// TIA Portal V16 export
// export: Created 2023-03-29T11:03:19.8804357Z, ExportSetting WithDefaults, DisplayName Totally Integrated Automation Portal, DisplayVersion V16 Update 6, DisplayName TIA Portal Version Control Interface, DisplayVersion V16 Update 2, DisplayName TIA Portal Openness, DisplayVersion V16 Update 6, DisplayName STEP 7 Professional, DisplayVersion V16 Update 6, DisplayName STEP 7 Safety, DisplayVersion V16, DisplayName WinCC Advanced, DisplayVersion V16 Update 6
DATA_BLOCK "DB10_instance_SCADA"   // DB10
TITLE = SCADA
{ S7_Optimized_Access := 'FALSE' }
AUTHOR : rtecmer
VERSION : 0.1
// stored: AutoNumber false, DBAccessibleFromOPCUA true, IsOnlyStoredInLoadMemory false, IsWriteProtectedInAS false
   VAR
      Clock : Time;
      Watchdog : Int;
      instZ1 : Word := 33924;   // status zasuwy
      instZ2 : Word := 33924;   // status zasuwy
      instZ3 : Word := 33924;   // status zasuwy
      instZ4 : Word := 33924;   // status zasuwy
      instZ5 : Word := 33924;   // status zasuwy
      instZ6 : Word := 33924;   // status zasuwy
      instZ7 : Word := 33924;   // status zasuwy
      instZ8 : Word := 33924;   // status zasuwy
      instZ9 : Word := 33924;   // status zasuwy
      instZ10 : Word := 33924;   // status zasuwy
      actPoziomZbiornik_1 : Real;   // aktualny poziom w zbirniku
      actPoziomZbiornik_2 : Real := 0.0;   // aktualny poziom w zbirniku
      actPoziomZbiornik_3 : Real := 0.0;   // aktualny poziom w zbirniku
      actPoziomZbiornik_4 : Real := 0.0;   // aktualny poziom w zbirniku
      actPoziomZbiornik_5 : Real := 0.0;   // aktualny poziom w zbirniku
      actPrzepływ_Q2 : Real;   // aktualny przepływ Q2 - studnia pomiarowa przed pompownią
      sumPrzepływVF_Q2 : Real;   // suma przepływu
      statusPrzepływVR_Q2 : Real := 0.0;   // status przepływomierza
      setPołożenieZ10 : Word := 40;   // zadany [%] otwarcia
      actPołożenieZ10 : Word;   // aktualny [%] otwarcia
      rtu_mpp04_2error_status : Word;   // status błędu modbus przepływomierz Q2
      ModelSterowania : Word;   // Sygnały sterowania strategią pompownia - 0= wyłaczone, 1=dosilanie, 2=przetłaczanie,3=automat, 4=ręczne
      TrybSterowania : Word;   // Tryb 0-wyłączony, 1- Dobowy, 2- Tygodniowy, 3-Ręczny
      "Alarms only" : Word;   // Instancja alarmów (bit 68.0 - Error komunikacji z HMI)
      setPoziomNapełniania : Real := 550.0;   // zadana wartość napełniania
      setPoziomOpróżnianai : Real := 30.0;   // zadana wartość opróżniania
      "actCiśnienie-magistralaB5" : Real := 6.6;   // ciśnienie na przewodzie zasilania 9magistrala)
      rtu_step_reset : Bool;   // reset modbus RTU
      actTime_FillingOn : Real;   // godzina start napełnianie
      actTime_FillingOff : Real;   // godzina stop napełnianie
      actTime_EptyingOn : Real;   // godzina start przetłaczanie
      actTime_EptyingOff : Real;   // godzina stop przetłaczanie
      actTime : Real;   // czas aktualny
      actDTL_FillingOn : DTL := DTL#2022-08-02-00:05:00;   // zmienna DTL napełnianie start
      actDTL_FillingOff : DTL := DTL#2022-08-02-17:00:00.000000003;   // zmienna DTL napełnianie stop
      actDTL_pumpingOn : DTL := DTL#2022-08-02-18:00:00.000000003;   // zmienna DTL przetłaczanie start
      actDTL_pumpingOff : DTL := DTL#2022-08-02-23:59:00.000000001;   // zmienna DTL przetłaczanie stop
      actDTL_RechargingOn : DTL := DTL#2022-08-02-18:00:00.000000013;   // zmienna DTL dosilanie start
      actDTL_RechargingOff : DTL := DTL#2022-08-02-23:59:00.000000003;   // zmienna DTL dosilanie stop
      reset_modbus_TCP : Bool;   // reset modbus TCP
      instConrol_ManAut_1 : Int := 0;   // Bity przełączenia trybu pracy napędów / 40019 Bity przełączenia trybu pracy napędów M1-M4, Zasuwami Z1, Z2, Z3, Z4
      instConrol_ManAut_2 : Int := 0;   // Bity przełączenia trybu pracy napędów / 40020 Bity przełączenia trybu pracy napędów Z5, Z6, Z7, Z8, Z9, Z10, Z11, Z12
   END_VAR
BEGIN
END_DATA_BLOCK
